FUNCTION_BLOCK MemoOC_D_HMI (* Service Interface Function Block Type *)
  (* Standard: 61499-2 *)
  (* Version 0.0, 6/7/2026, Schneider Electric, template *)
  PACKAGE SE.Nereda;
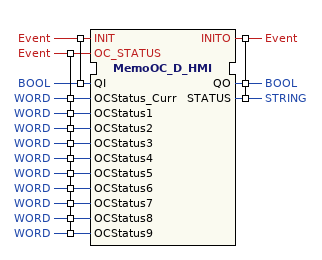
  EVENT_INPUT
    INIT WITH QI;
    OC_STATUS WITH OCStatus_Curr, OCStatus1, OCStatus2, OCStatus3, OCStatus4, OCStatus5, OCStatus6, OCStatus7, OCStatus8, OCStatus9;
  END_EVENT
  EVENT_OUTPUT
    INITO WITH QO, STATUS;
  END_EVENT
  VAR_INPUT
    QI : BOOL;
    OCStatus_Curr : WORD;
    OCStatus1 : WORD;
    OCStatus2 : WORD;
    OCStatus3 : WORD;
    OCStatus4 : WORD;
    OCStatus5 : WORD;
    OCStatus6 : WORD;
    OCStatus7 : WORD;
    OCStatus8 : WORD;
    OCStatus9 : WORD;
  END_VAR
  VAR_OUTPUT
    QO : BOOL; (* Event Output Qualifier *)
    STATUS : STRING; (* Service Status *)
  END_VAR
  SERVICE /
    SEQUENCE 
    END_SEQUENCE
  END_SERVICE
END_FUNCTION_BLOCK
